// LS Electric XG5000 project: TMR
// PLC LSPLC
// module base 0 slot 0: 입출력 모듈:XBC-DR30S (DC 24V 입력 18점, 릴레이 출력 12점)

PROGRAM TMR (task: 스캔 프로그램)

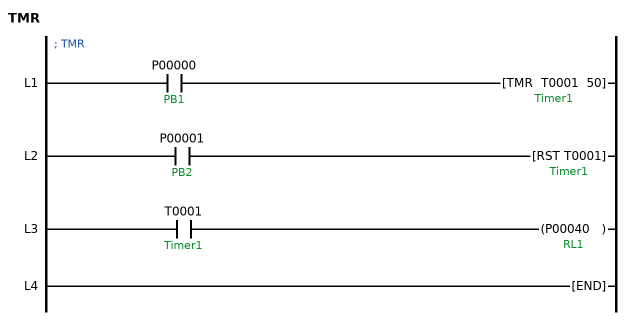
// TMR
; L1
LOAD      P00000	// PB1
TMR       T0001 50	// Timer1
; L2
LOAD      P00001	// PB2
RST       T0001	// Timer1
; L3
LOAD      T0001	// Timer1
OUT       P00040	// RL1
; L4
END